FUNCTION_BLOCK PAFMixing EXTENDS PAProcessFunction IMPLEMENTS IPAFMixing
VAR_INPUT
END_VAR
VAR_OUTPUT
END_VAR
VAR
	_ACMethod : ACMethodMixing;
END_VAR

PROPERTY ACMethod : IACMethod
GET
ACMethod := _ACMethod;
END_GET
END_PROPERTY

METHOD PROTECTED SMIdle
VAR_INPUT
END_VAR
SUPER^.SMIdle();
END_METHOD

METHOD PUBLIC StartWithP : BOOL
VAR_INPUT
	parameter : ACMethodMixingP;
END_VAR
VAR
	acMethod : ACMethodMixing;
END_VAR
acMethod.Parameter := parameter;
IF NOT acMethod.IsValid THEN
		StartWithP := FALSE;
	RETURN;
END_IF
_ACMethod.Parameter := parameter;
StartWithP := Start();
END_METHOD

END_FUNCTION_BLOCK

(* stored: Version 1.1.0.1, ProductVersion 3.1.4020.12
   POU PAFMixing: Id {fcd6110b-9e7e-460f-9a0e-7bc2ea8862dc}, SpecialFunc None
   Folder StateMethods: Id {c6ae6d40-1f86-48f4-ab74-575284abfa17}
   Property ACMethod: Id {dccc899c-3d03-4086-8c03-3b0b8f0ad21b}
   Get Get: Id {f3fd84a5-61eb-4114-a83b-103fb15caddb}
   Method SMIdle: Id {8ee9f5fa-571d-4f3e-8ce3-a318338e467b}
   Method StartWithP: Id {28ce06cf-d91b-41b1-89a0-b612b40ea290} *)
